PROGRAM P_DimmingLight_Test_CFC
VAR
	fbDimmingLight		:	FB_DimmingLight;
	bOn					:	BOOL;
	bOff				:	BOOL;
	bRecallMinLevel		:	BOOL;
	bSetControlLevel	:	BOOL;
	nSetControlLevel	:	BYTE;
	bControlLevel		:	BOOL;
	nControlLevel		:	BYTE;
END_VAR

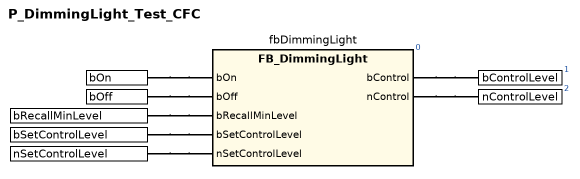
fbDimmingLight(
    bOn := bOn,
    bOff := bOff,
    bRecallMinLevel := bRecallMinLevel,
    bSetControlLevel := bSetControlLevel,
    nSetControlLevel := nSetControlLevel); // FB_DimmingLight
bControlLevel := fbDimmingLight.bControl;
nControlLevel := fbDimmingLight.nControl;

END_PROGRAM

(* stored: Version 1.1.0.1, ProductVersion 3.1.0.23
   POU P_DimmingLight_Test_CFC: Id {19678740-a9f2-4c9d-a3af-951aff7688dc} *)
